FUNCTION_BLOCK GreenMasterDO EXTENDS GreenMasterDO_Base
VAR_INPUT
END_VAR
VAR_OUTPUT
END_VAR
VAR_IN_OUT
END_VAR
VAR
	IO_DO_01: DigitalOutput;
	IO_DO_02: DigitalOutput;
	IO_DO_03: DigitalOutput;
	IO_DO_04: DigitalOutput;
	IO_DO_05: DigitalOutput;
	IO_DO_06: DigitalOutput;
	IO_DO_07: DigitalOutput;
	IO_DO_08: DigitalOutput;
	IO_DO_09: DigitalOutput;
	IO_DO_10: DigitalOutput;
	IO_DO_11: DigitalOutput;
	IO_DO_12: DigitalOutput;
	IO_DO_13: DigitalOutput;
	IO_DO_14: DigitalOutput;
	IO_RDO_01: DigitalOutput;
	IO_RDO_02: DigitalOutput;
	IO_RDO_03: DigitalOutput;
	IO_RDO_04: DigitalOutput;
	IO_DO_16: DigitalOutput;
END_VAR


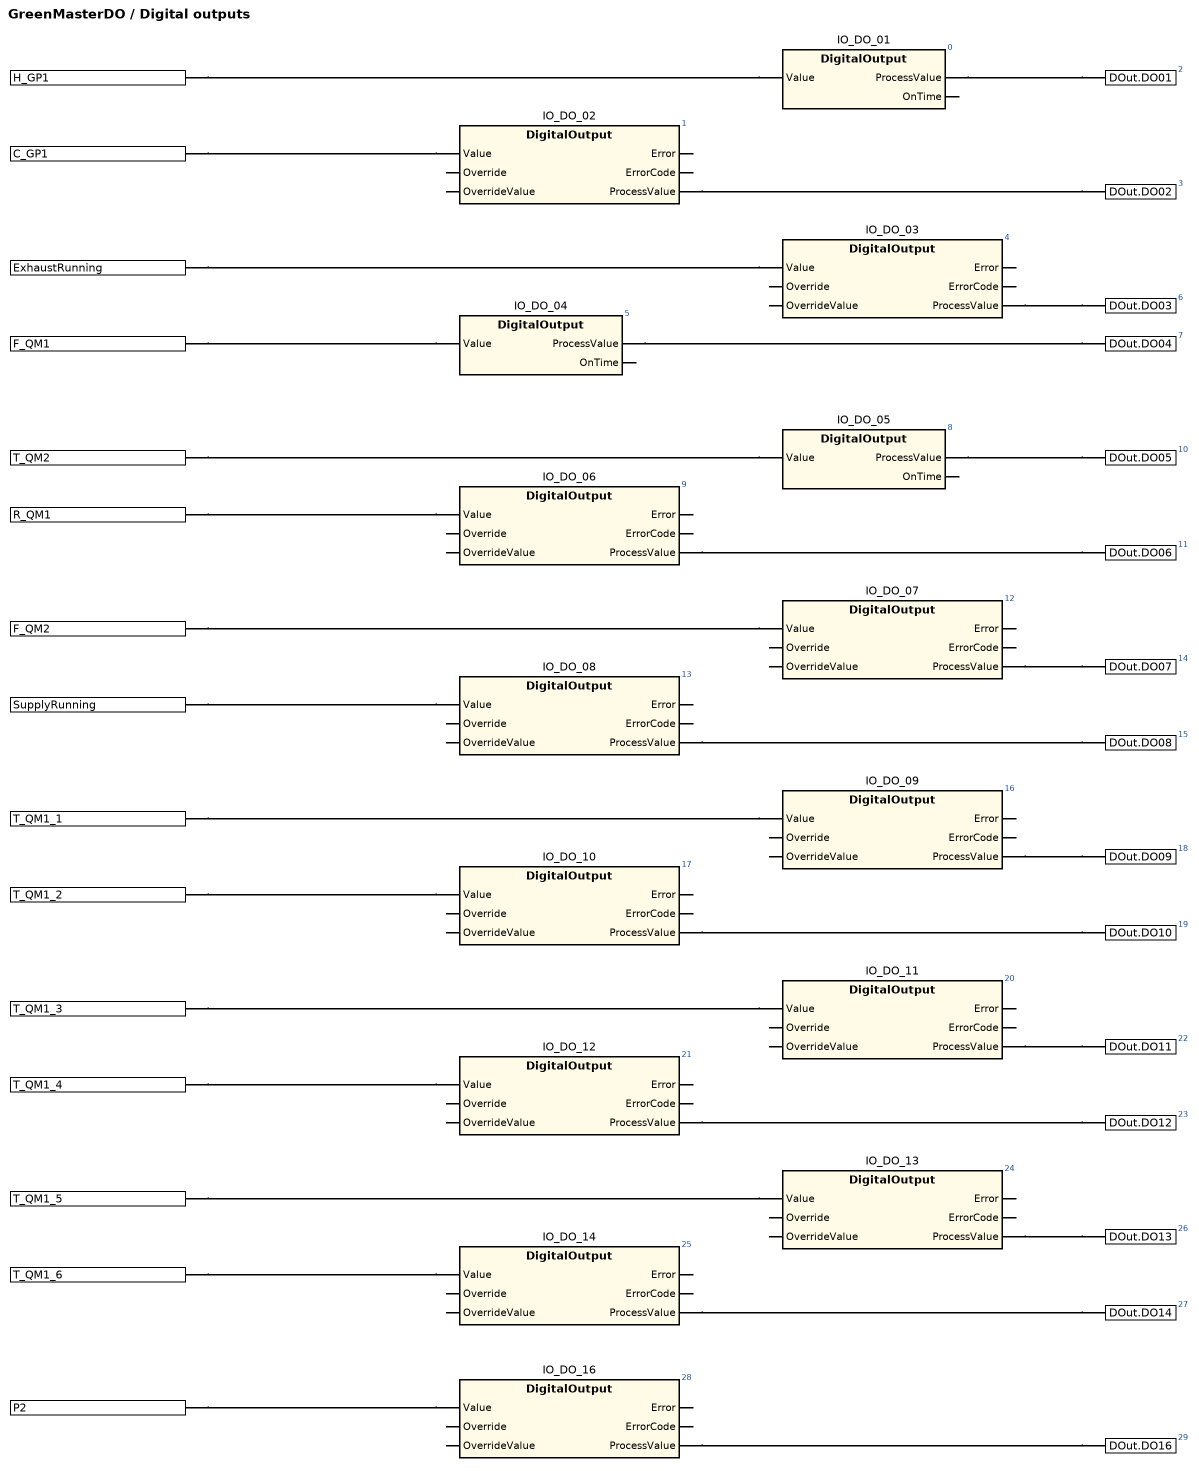
// PAGE Digital outputs
IO_DO_01(Value := H_GP1); // DigitalOutput
IO_DO_02(Value := C_GP1); // DigitalOutput
DOut.DO01 := IO_DO_01.ProcessValue;
DOut.DO02 := IO_DO_02.ProcessValue;
IO_DO_03(Value := ExhaustRunning); // DigitalOutput
IO_DO_04(Value := F_QM1); // DigitalOutput
DOut.DO03 := IO_DO_03.ProcessValue;
DOut.DO04 := IO_DO_04.ProcessValue;
IO_DO_05(Value := T_QM2); // DigitalOutput
IO_DO_06(Value := R_QM1); // DigitalOutput
DOut.DO05 := IO_DO_05.ProcessValue;
DOut.DO06 := IO_DO_06.ProcessValue;
IO_DO_07(Value := F_QM2); // DigitalOutput
IO_DO_08(Value := SupplyRunning); // DigitalOutput
DOut.DO07 := IO_DO_07.ProcessValue;
DOut.DO08 := IO_DO_08.ProcessValue;
IO_DO_09(Value := T_QM1_1); // DigitalOutput
IO_DO_10(Value := T_QM1_2); // DigitalOutput
DOut.DO09 := IO_DO_09.ProcessValue;
DOut.DO10 := IO_DO_10.ProcessValue;
IO_DO_11(Value := T_QM1_3); // DigitalOutput
IO_DO_12(Value := T_QM1_4); // DigitalOutput
DOut.DO11 := IO_DO_11.ProcessValue;
DOut.DO12 := IO_DO_12.ProcessValue;
IO_DO_13(Value := T_QM1_5); // DigitalOutput
IO_DO_14(Value := T_QM1_6); // DigitalOutput
DOut.DO13 := IO_DO_13.ProcessValue;
DOut.DO14 := IO_DO_14.ProcessValue;
IO_DO_16(Value := P2); // DigitalOutput
DOut.DO16 := IO_DO_16.ProcessValue;

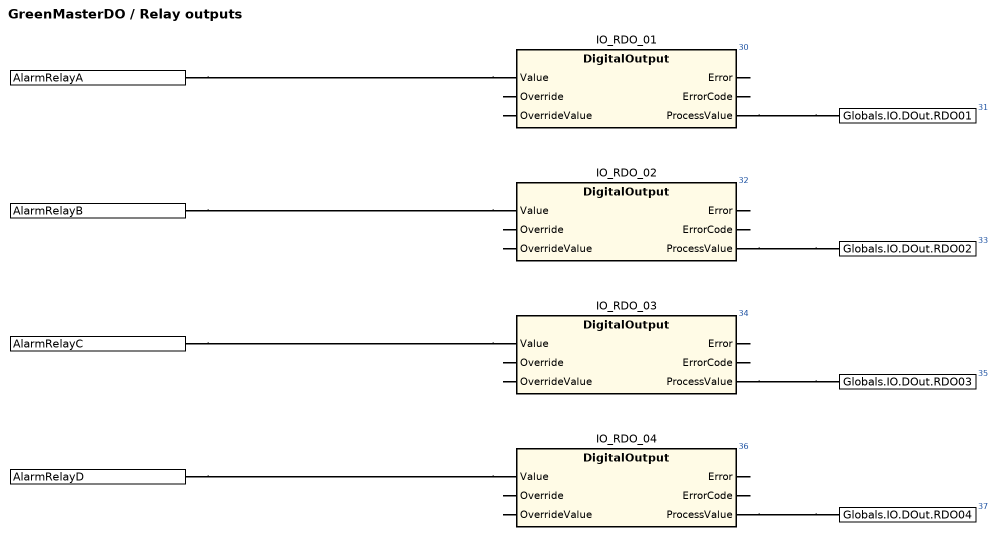
// PAGE Relay outputs
IO_RDO_01(Value := AlarmRelayA); // DigitalOutput
Globals.IO.DOut.RDO01 := IO_RDO_01.ProcessValue;
IO_RDO_02(Value := AlarmRelayB); // DigitalOutput
Globals.IO.DOut.RDO02 := IO_RDO_02.ProcessValue;
IO_RDO_03(Value := AlarmRelayC); // DigitalOutput
Globals.IO.DOut.RDO03 := IO_RDO_03.ProcessValue;
IO_RDO_04(Value := AlarmRelayD); // DigitalOutput
Globals.IO.DOut.RDO04 := IO_RDO_04.ProcessValue;

METHOD SetOverrides : BOOL
VAR_INPUT
	Override: DigitalOutputOverrideParameters;
END_VAR
IF Main.ManualAllowed THEN
	IO_DO_01.Override := Override.H_GP1_Override;
	IO_DO_01.OverrideValue := Override.H_GP1_OverrideValue;
	IO_DO_02.Override := Override.C_GP1_Override;
	IO_DO_02.OverrideValue := Override.C_GP1_OverrideValue;
	IO_DO_03.Override := Override.F_RUN_Override;
	IO_DO_03.OverrideValue := Override.F_RUN_OverrideValue;
	IO_DO_04.Override := Override.F_QM1_Override;
	IO_DO_04.OverrideValue := Override.F_QM1_OverrideValue;
	IO_DO_05.Override := Override.T_QM2_Override;
	IO_DO_05.OverrideValue := Override.T_QM2_OverrideValue;
	IO_DO_06.Override := Override.R_QM1_Override;
	IO_DO_06.OverrideValue := Override.R_QM1_OverrideValue;
	IO_DO_07.Override := Override.F_QM2_Override;
	IO_DO_07.OverrideValue := Override.F_QM2_OverrideValue;
	IO_DO_08.Override := Override.T_RUN_Override;
	IO_DO_08.OverrideValue := Override.T_RUN_OverrideValue;
	IO_DO_09.Override := Override.T_QM1_1_Override;
	IO_DO_09.OverrideValue := Override.T_QM1_1_OverrideValue;
	IO_DO_10.Override := Override.T_QM1_2_Override;
	IO_DO_10.OverrideValue := Override.T_QM1_2_OverrideValue;
	IO_DO_11.Override := Override.T_QM1_3_Override;
	IO_DO_11.OverrideValue := Override.T_QM1_3_OverrideValue;
	IO_DO_12.Override := Override.T_QM1_4_Override;
	IO_DO_12.OverrideValue := Override.T_QM1_4_OverrideValue;
	IO_DO_13.Override := Override.T_QM1_5_Override;
	IO_DO_13.OverrideValue := Override.T_QM1_5_OverrideValue;
	IO_DO_14.Override := Override.T_QM1_6_Override;
	IO_DO_14.OverrideValue := Override.T_QM1_6_OverrideValue;
	IO_DO_16.Override := Override.P2_Override;
	IO_DO_16.OverrideValue := Override.P2_OverrideValue;
ELSE	
	IO_DO_01.Override := FALSE;
	IO_DO_02.Override := FALSE;
	IO_DO_03.Override := FALSE;
	IO_DO_04.Override := FALSE;
	IO_DO_05.Override := FALSE;
	IO_DO_06.Override := FALSE;
	IO_DO_07.Override := FALSE;
	IO_DO_08.Override := FALSE;
	IO_DO_09.Override := FALSE;
	IO_DO_10.Override := FALSE;
	IO_DO_11.Override := FALSE;
	IO_DO_12.Override := FALSE;
	IO_DO_13.Override := FALSE;
	IO_DO_14.Override := FALSE;
	IO_DO_16.Override := FALSE;
END_IF
END_METHOD

END_FUNCTION_BLOCK

(* stored: Version 1.1.0.1, ProductVersion 3.1.4024.6
   POU GreenMasterDO: Id {239f4845-259c-4ac2-815a-224d60d0147b}, SpecialFunc None
   Method SetOverrides: Id {09b97b0e-cefc-4c0c-b961-435325ba9e9d} *)
